// Mitsubishi GX Works2 project: SelfHolding   PLC: Q03UDV

PROGRAM MAIN
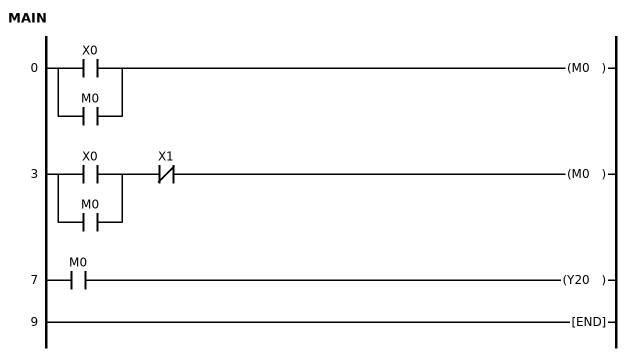
0     LD      X0
      OR      M0
      OUT     M0
3     LD      X0
      OR      M0
      ANI     X1
      OUT     M0
7     LD      M0
      OUT     Y20
9     END
END_PROGRAM
